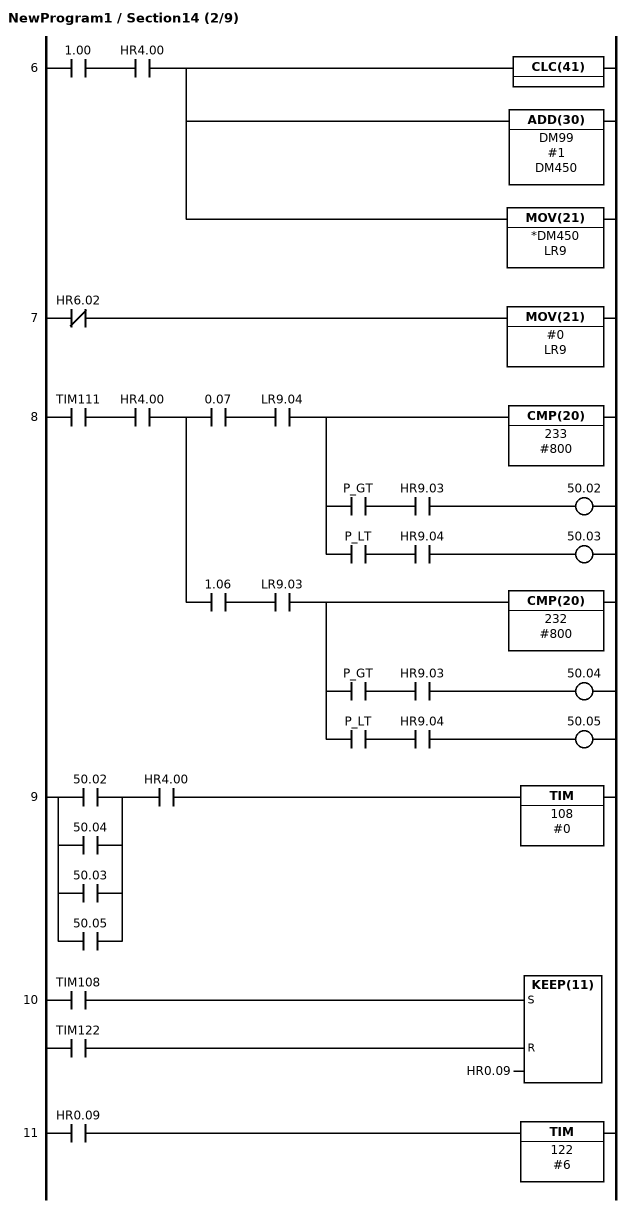
; [picture p72: NewProgram1 / Section14, rungs 6-11]
; rung 6
LD 1.00
AND HR4.00
CLC(41)
ADD(30) DM99 #1 DM450
MOV(21) *DM450 LR9
; rung 7
LDNOT HR6.02
MOV(21) #0 LR9
; rung 8
LD TIM111
AND HR4.00
OUT TR0
AND 0.07
AND LR9.04
OUT TR1
CMP(20) 233 #800
AND P_GT
AND HR9.03
OUT 50.02
LD TR1
AND P_LT
AND HR9.04
OUT 50.03
LD TR0
AND 1.06
AND LR9.03
OUT TR0
CMP(20) 232 #800
AND P_GT
AND HR9.03
OUT 50.04
LD TR0
AND P_LT
AND HR9.04
OUT 50.05
; rung 9
LD 50.02
OR 50.04
OR 50.03
OR 50.05
AND HR4.00
TIM 108 #0
; rung 10
LD TIM108
LD TIM122
KEEP(11) HR0.09
; rung 11
LD HR0.09
TIM 122 #6

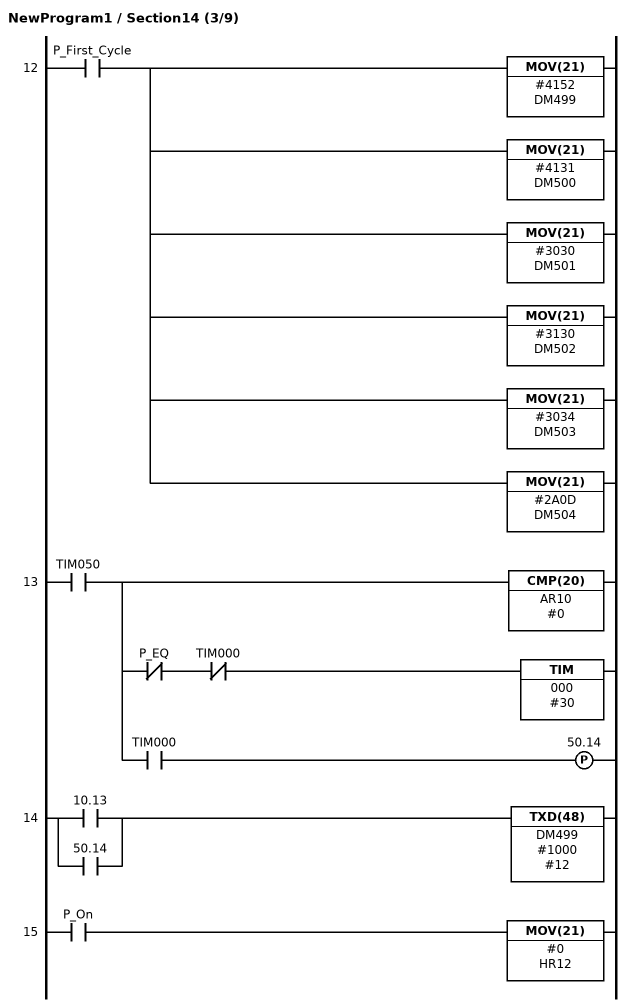
; rung 12
LD P_First_Cycle
MOV(21) #4152 DM499
MOV(21) #4131 DM500
MOV(21) #3030 DM501
MOV(21) #3130 DM502
MOV(21) #3034 DM503
MOV(21) #2A0D DM504
; rung 13
LD TIM050
OUT TR0
CMP(20) AR10 #0
ANDNOT P_EQ
ANDNOT TIM000
TIM 000 #30
LD TR0
AND TIM000
DIFU(13) 50.14
; rung 14
LD 10.13
OR 50.14
TXD(48) DM499 #1000 #12
; rung 15
LD P_On
MOV(21) #0 HR12

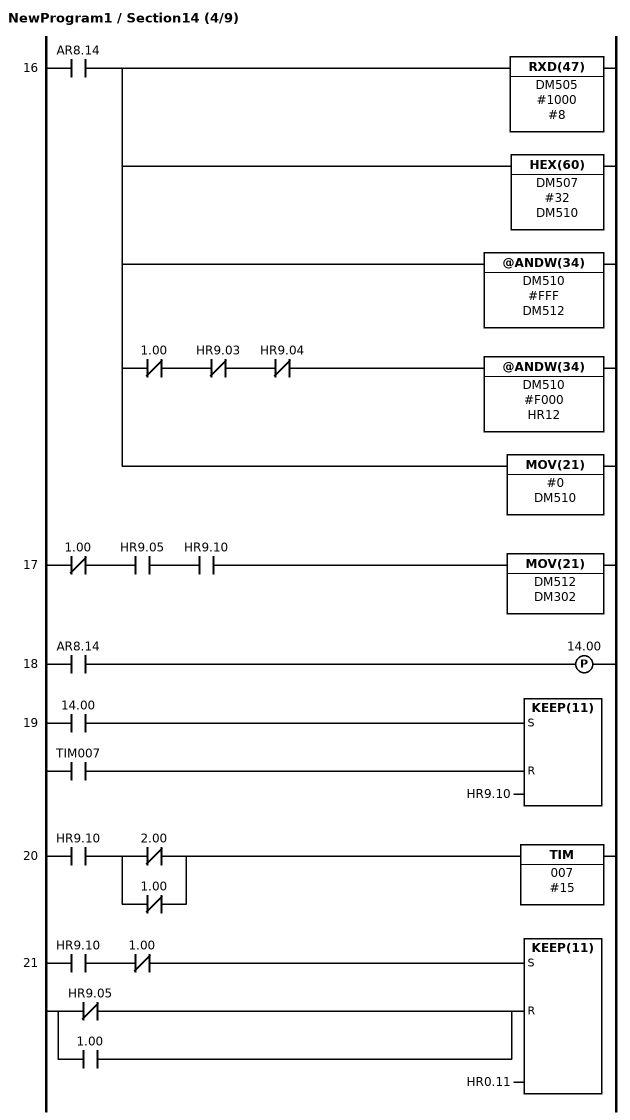
; rung 16
LD AR8.14
OUT TR0
RXD(47) DM505 #1000 #8
HEX(60) DM507 #32 DM510
@ANDW(34) DM510 #FFF DM512
ANDNOT 1.00
ANDNOT HR9.03
ANDNOT HR9.04
@ANDW(34) DM510 #F000 HR12
LD TR0
MOV(21) #0 DM510
; rung 17
LDNOT 1.00
AND HR9.05
AND HR9.10
MOV(21) DM512 DM302
; rung 18
LD AR8.14
DIFU(13) 14.00
; rung 19
LD 14.00
LD TIM007
KEEP(11) HR9.10
; rung 20
LD HR9.10
LDNOT 2.00
ORNOT 1.00
ANDLD
TIM 007 #15
; rung 21
LD HR9.10
ANDNOT 1.00
LDNOT HR9.05
OR 1.00
KEEP(11) HR0.11

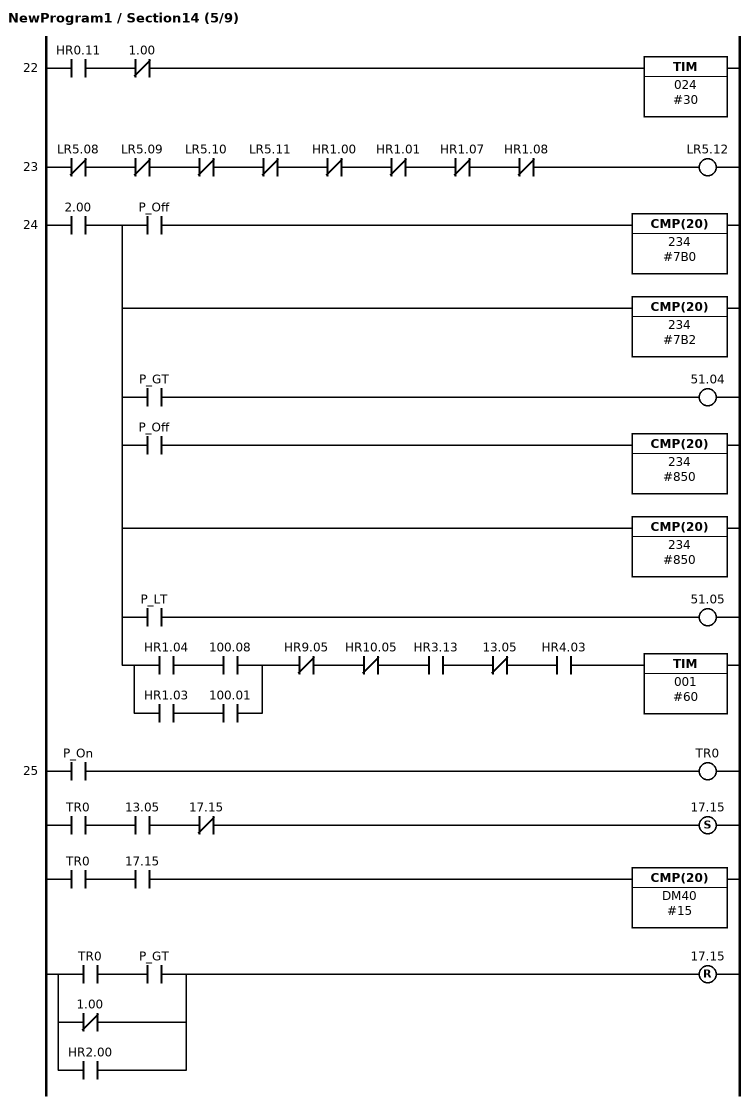
; rung 22
LD HR0.11
ANDNOT 1.00
TIM 024 #30
; rung 23
LDNOT LR5.08
ANDNOT LR5.09
ANDNOT LR5.10
ANDNOT LR5.11
ANDNOT HR1.00
ANDNOT HR1.01
ANDNOT HR1.07
ANDNOT HR1.08
OUT LR5.12
; rung 24
LD 2.00
OUT TR0
AND P_Off
CMP(20) 234 #7B0
LD TR0
CMP(20) 234 #7B2
AND P_GT
OUT 51.04
LD TR0
AND P_Off
CMP(20) 234 #850
LD TR0
CMP(20) 234 #850
AND P_LT
OUT 51.05
LD TR0
LD HR1.04
AND 100.08
LD HR1.03
AND 100.01
ORLD
ANDLD
ANDNOT HR9.05
ANDNOT HR10.05
AND HR3.13
ANDNOT 13.05
AND HR4.03
TIM 001 #60
; rung 25
LD P_On
OUT TR0
AND 13.05
ANDNOT 17.15
SET 17.15
LD TR0
AND 17.15
CMP(20) DM40 #15
LD TR0
AND P_GT
LDNOT 1.00
OR HR2.00
ORLD
RSET 17.15

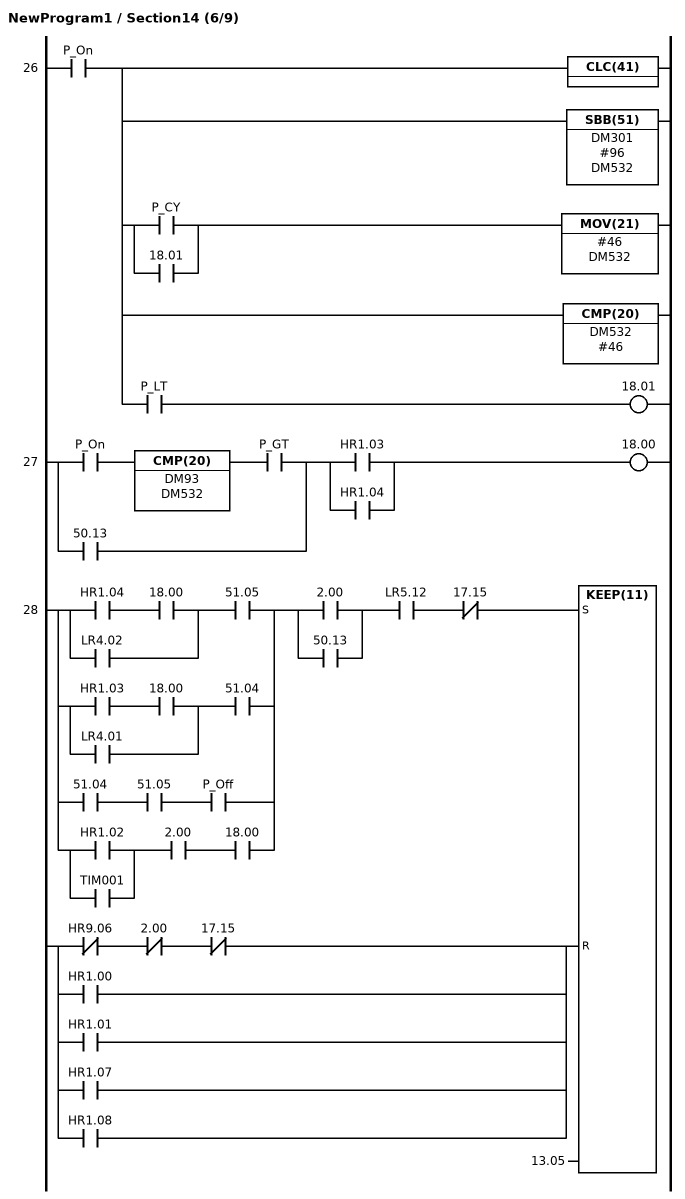
; rung 26
LD P_On
OUT TR0
CLC(41)
SBB(51) DM301 #96 DM532
LD P_CY
OR 18.01
ANDLD
MOV(21) #46 DM532
LD TR0
CMP(20) DM532 #46
AND P_LT
OUT 18.01
; rung 27
LD P_On
CMP(20) DM93 DM532
AND P_GT
OR 50.13
LD HR1.03
OR HR1.04
ANDLD
OUT 18.00
; rung 28
LD HR1.04
AND 18.00
OR LR4.02
AND 51.05
LD HR1.03
AND 18.00
OR LR4.01
AND 51.04
ORLD
LD 51.04
AND 51.05
AND P_Off
ORLD
LD HR1.02
OR TIM001
AND 2.00
AND 18.00
ORLD
LD 2.00
OR 50.13
ANDLD
AND LR5.12
ANDNOT 17.15
LDNOT HR9.06
ANDNOT 2.00
ANDNOT 17.15
OR HR1.00
OR HR1.01
OR HR1.07
OR HR1.08
KEEP(11) 13.05

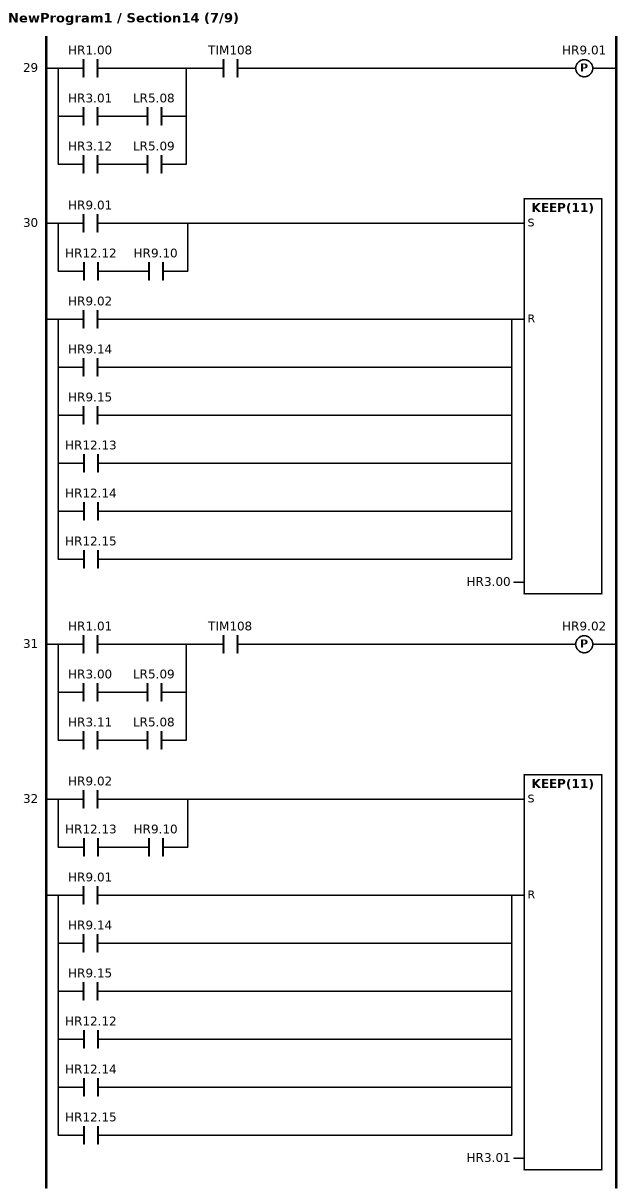
; rung 29
LD HR1.00
LD HR3.01
AND LR5.08
ORLD
LD HR3.12
AND LR5.09
ORLD
AND TIM108
DIFU(13) HR9.01
; rung 30
LD HR9.01
LD HR12.12
AND HR9.10
ORLD
LD HR9.02
OR HR9.14
OR HR9.15
OR HR12.13
OR HR12.14
OR HR12.15
KEEP(11) HR3.00
; rung 31
LD HR1.01
LD HR3.00
AND LR5.09
ORLD
LD HR3.11
AND LR5.08
ORLD
AND TIM108
DIFU(13) HR9.02
; rung 32
LD HR9.02
LD HR12.13
AND HR9.10
ORLD
LD HR9.01
OR HR9.14
OR HR9.15
OR HR12.12
OR HR12.14
OR HR12.15
KEEP(11) HR3.01

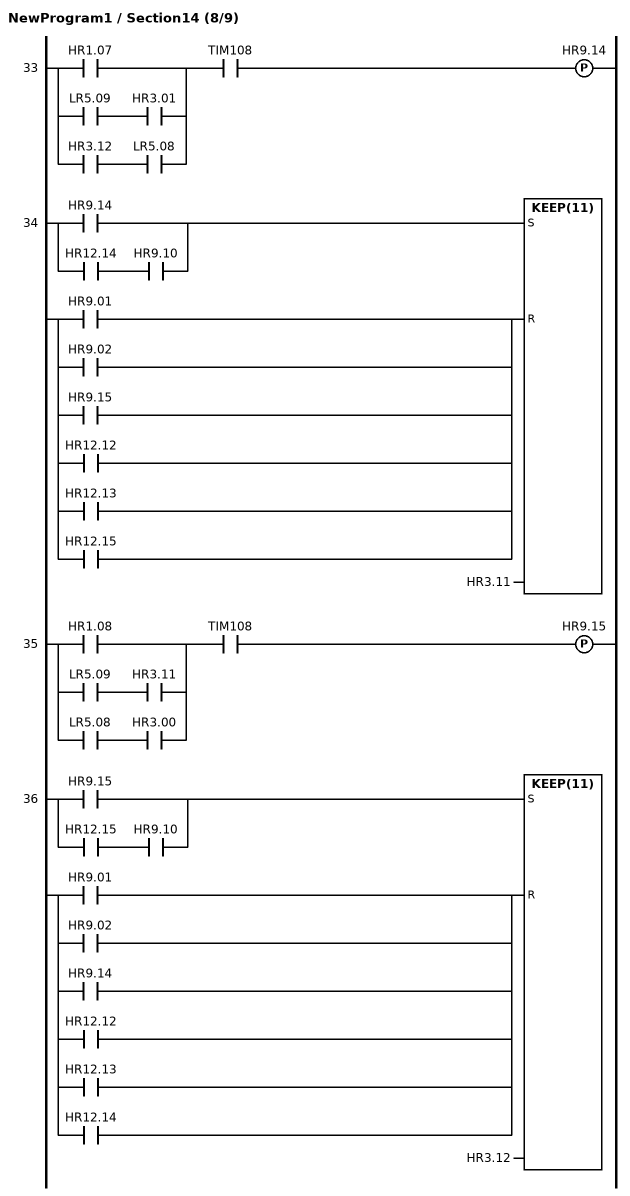
; rung 33
LD HR1.07
LD LR5.09
AND HR3.01
ORLD
LD HR3.12
AND LR5.08
ORLD
AND TIM108
DIFU(13) HR9.14
; rung 34
LD HR9.14
LD HR12.14
AND HR9.10
ORLD
LD HR9.01
OR HR9.02
OR HR9.15
OR HR12.12
OR HR12.13
OR HR12.15
KEEP(11) HR3.11
; rung 35
LD HR1.08
LD LR5.09
AND HR3.11
ORLD
LD LR5.08
AND HR3.00
ORLD
AND TIM108
DIFU(13) HR9.15
; rung 36
LD HR9.15
LD HR12.15
AND HR9.10
ORLD
LD HR9.01
OR HR9.02
OR HR9.14
OR HR12.12
OR HR12.13
OR HR12.14
KEEP(11) HR3.12

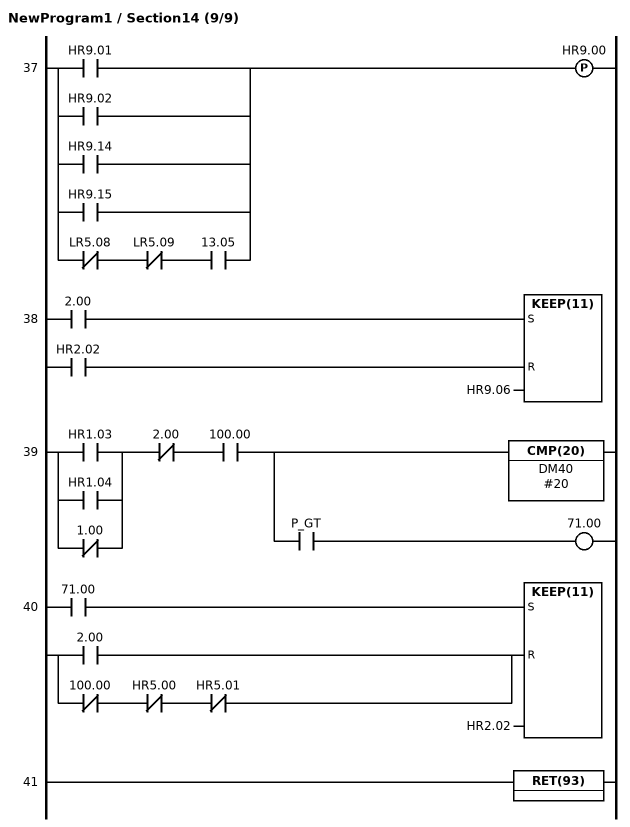
; rung 37
LD HR9.01
OR HR9.02
OR HR9.14
OR HR9.15
LDNOT LR5.08
ANDNOT LR5.09
AND 13.05
ORLD
DIFU(13) HR9.00
; rung 38
LD 2.00
LD HR2.02
KEEP(11) HR9.06
; rung 39
LD HR1.03
OR HR1.04
ORNOT 1.00
ANDNOT 2.00
AND 100.00
CMP(20) DM40 #20
AND P_GT
OUT 71.00
; rung 40
LD 71.00
LD 2.00
LDNOT 100.00
ANDNOT HR5.00
ANDNOT HR5.01
ORLD
KEEP(11) HR2.02
; rung 41
RET(93)

### Section Section15

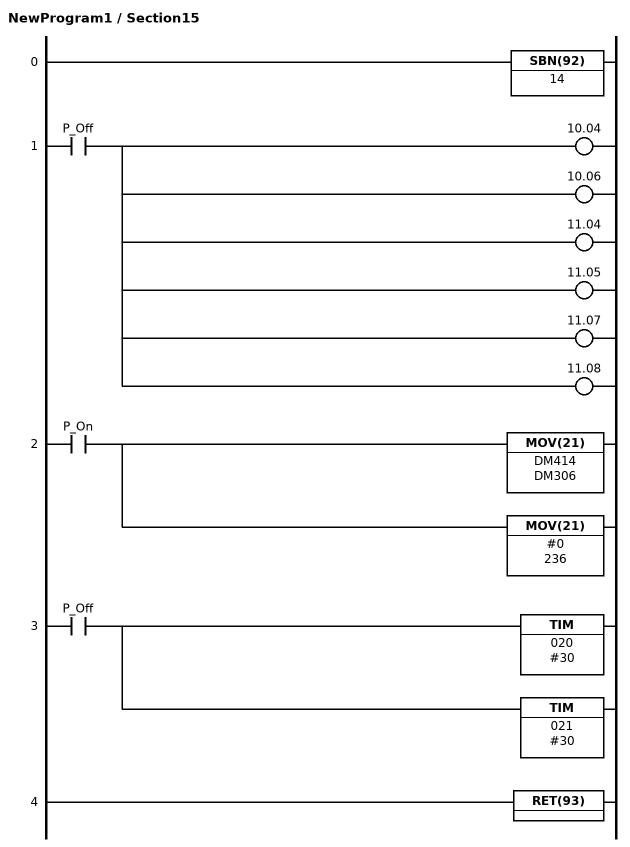
; rung 0
SBN(92) 14
; rung 1
LD P_Off
OUT 10.04
OUT 10.06
OUT 11.04
OUT 11.05
OUT 11.07
OUT 11.08
; rung 2
LD P_On
MOV(21) DM414 DM306
MOV(21) #0 236
; rung 3
LD P_Off
TIM 020 #30
TIM 021 #30
; rung 4
RET(93)

### Section Section16

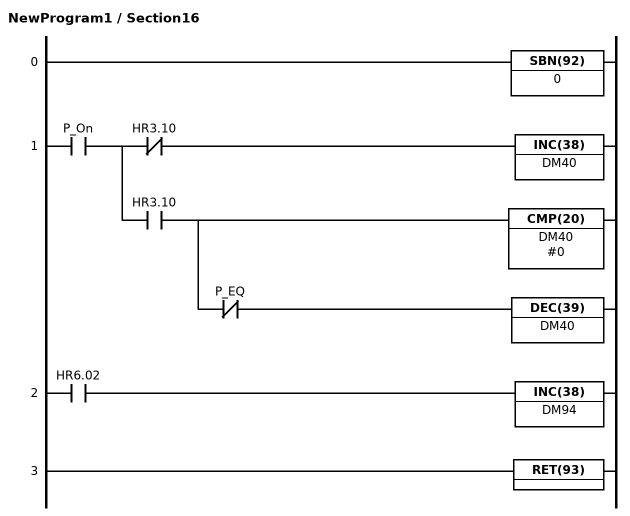
; rung 0
SBN(92) 0
; rung 1
LD P_On
OUT TR0
ANDNOT HR3.10
INC(38) DM40
LD TR0
AND HR3.10
CMP(20) DM40 #0
ANDNOT P_EQ
DEC(39) DM40
; rung 2
LD HR6.02
INC(38) DM94
; rung 3
RET(93)

### Section Section17
; rung 0
END(01)